// SIMATIC S7-200 project (STEP 7-Micro/WIN), CPU 224XP REL 02.01

SYMBOL_TABLE USUARIO1
P_SUBIR          I0.0
P_BAJAR          I0.1
P_DERECHA        I0.2
P_IIZQUIERDA     I0.3
FC_ABAJO         I0.4
FC_ARRIBA        I0.5
FC_IZQUIERDA     I0.6
FC_DERECHA       I0.7
M1_SUBIR         Q0.0
M1_BAJAR         Q0.1
M2_IZQUIERDA     Q0.2
M2_DERECHA       Q0.3
END_SYMBOL_TABLE

ORGANIZATION_BLOCK PRINCIPAL:OB1
TITLE=COMENTARIOS DEL PROGRAMA
BEGIN
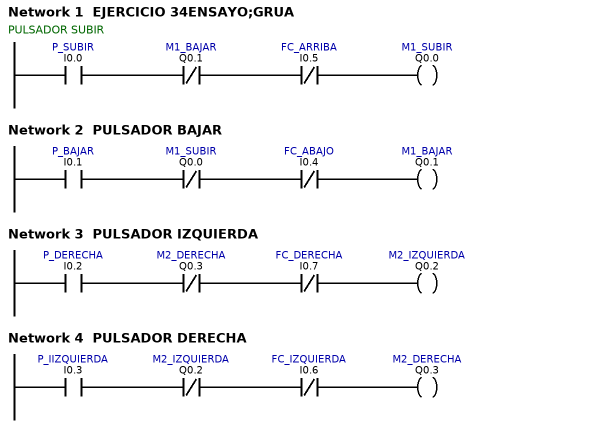
Network 1 // EJERCICIO 34ENSAYO;GRUA
 
// PULSADOR SUBIR
// (network saved uncompiled; LAD cells follow)
// row 0: c0 -| |- P_SUBIR:I0.0  c1 -|/|- M1_BAJAR:Q0.1  c2 -|/|- FC_ARRIBA:I0.5  c3 -( ) M1_SUBIR:Q0.0
Network 2 // PULSADOR BAJAR
// (network saved uncompiled; LAD cells follow)
// row 0: c0 -| |- P_BAJAR:I0.1  c1 -|/|- M1_SUBIR:Q0.0  c2 -|/|- FC_ABAJO:I0.4  c3 -( ) M1_BAJAR:Q0.1
Network 3 // PULSADOR IZQUIERDA
// (network saved uncompiled; LAD cells follow)
// row 0: c0 -| |- P_DERECHA:I0.2  c1 -|/|- M2_DERECHA:Q0.3  c2 -|/|- FC_DERECHA:I0.7  c3 -( ) M2_IZQUIERDA:Q0.2
Network 4 // PULSADOR DERECHA 
// (network saved uncompiled; LAD cells follow)
// row 0: c0 -| |- P_IIZQUIERDA:I0.3  c1 -|/|- M2_IZQUIERDA:Q0.2  c2 -|/|- FC_IZQUIERDA:I0.6  c3 -( ) M2_DERECHA:Q0.3
END_ORGANIZATION_BLOCK
